EQUP_TYPE_1_Pump_RB(
	i1:= NOT( reactorB1.q6 AND reactorB2.q6 AND reactorB3.q6 AND reactorB4.q6),
	i2:= reactorB1.q6 OR reactorB2.q6 OR reactorB3.q6 OR reactorB4.q6,
	r1:= reset_Pump2_RB,
	sa1:=P201B1_DesludgePumpS2_EStopStat ,
	sa2:= ,
	sa3:=P201B1_DesludgePumpS2_LocalRemoteStat ,
	sa4:= P201B1_DesludgePumpS2_OverloadStat,
	sa5:=P201B1_DesludgePumpS2_RunStat ,
	sb1:= P201B2_DesludgePumpS2_EStopStat,
	sb2:= ,
	sb3:=P201B2_DesludgePumpS2_LocalRemoteStat ,
	sb4:= P201B2_DesludgePumpS2_OverloadStat,
	sb5:=P201B2_DesludgePumpS2_RunStat ,
	c1=> ,
	c2=> ,
	q1=>P201B1_DesludgePumpS2_RunCmd,
	q2=>P201B2_DesludgePumpS2_RunCmd ,
	e1=> );


EQUIP_TYPE_3_Valva1_RB1(
	i1:=NOT reactorB1.q1 ,
	i2:=reactorB1.q1 ,
	s1:=XV205B_SBRValveR1_CloseStat ,
	s2:=XV205B_SBRValveR1_OpenStat ,
	c1=> ,
	q1=>XV205B_SBRValveR1_CloseCmd ,
	q2=>XV205B_SBRValveR1_OpenCmd);

EQUIP_TYPE_8_MIXER_B1(
	i1:= NOT reactorB1.q2,
	i2:= reactorB1.q2,
	sa1:=M200B1A_MixerR1_EStopStat,
	sa2:=M200B1A_MixerR1_IncompleteStat ,
	sa3:=M200B1A_MixerR1_LocalRemoteStat ,
	sa4:=M200B1A_MixerR1_OverloadStat ,
	sa5:=M200B1A_MixerR1_RunStat ,
	sb1:=M200B1B_MixerR1_EStopStat,
	sb2:=M200B1B_MixerR1_IncompleteStat ,
	sb3:=M200B1B_MixerR1_LocalRemoteStat ,
	sb4:=M200B1B_MixerR1_OverloadStat ,
	sb5:=M200B1B_MixerR1_RunStat ,
	sc1:=M200B1C_MixerR1_EStopStat,
	sc2:=M200B1C_MixerR1_IncompleteStat ,
	sc3:=M200B1C_MixerR1_LocalRemoteStat ,
	sc4:=M200B1C_MixerR1_OverloadStat ,
	sc5:=M200B1C_MixerR1_RunStat ,
	c1=> ,
	q1=>M200B1A_MixerR1_RunCmd ,
	q2=>M200B1B_MixerR1_RunCmd,
	q3=>M200B1C_MixerR1_RunCmd ,
	e1=> );

EQUIP_TYPE_3_Valve2_RB1(
	i1:=NOT reactorB1.q3 ,
	i2:= reactorB1.q3,
	s1:= XV221B_LimeValveR1_CloseStat,
	s2:= XV221B_LimeValveR1_OpenStat,
	c1=> ,
	q1=>XV221B_LimeValveR1_CloseCmd ,
	q2=>XV221B_LimeValveR1_OpenCmd );

EQUIP_TYPE_3_Valve3_RB1(
	i1:=NOT reactorB1.q4 ,
	i2:= reactorB1.q4,
	s1:= XV211B_AlumValveR1_CloseStat,
	s2:= XV211B_AlumValveR1_OpenStat,
	c1=> ,
	q1=>XV211B_AlumValveR1_CloseCmd ,
	q2=>XV211B_AlumValveR1_OpenCmd );

EQUIP_TYPE_3_Valve4_RB1(
	i1:=NOT reactorB1.q5 ,
	i2:= reactorB1.q5,
	s1:=XV201B_AirBlowerValveR1_CloseStat ,
	s2:=XV201B_AirBlowerValveR1_OpenStat ,
	c1=> ,
	q1=>XV201B_AirBlowerValveR1_CloseCmd ,
	q2=>XV201B_AirBlowerValveR1_OpenCmd );

EQUIP_TYPE_9_Valve5_RB1(
	i1:= NOT reactorB1.q7 ,
	i2:=reactorB1.q7 ,
	(*s1:=XV241B_SludgeValveR1_CloseStat ,*)
	(*s2:=XV241B_SludgeValveR1_OpenStat ,*)
	c1=> ,
	q1=>XV241B_SludgeValveR1_CloseCmd ,
	q2=>XV241B_SludgeValveR1_OpenCmd );

EQUIP_TYPE_10_Dec_RB1(
	i1:=reactorB1.q8 ,
	i2:= reactorB1.q9,
	r1:= reset_dec_RB1,
	s1:= XV261B_DecanterR1_EStopStat,
	s2:= XV261B_DecanterR1_FwdStat,
	s3:= XV261B_DecanterR1_OverloadStat,
	s4:= XV261B_DecanterR1_OverloadStat,
	s5:= XV261B_DecanterR1_RvsStat,
	q1=> XV261B_DecanterR1_RvsCmd,
	q2=>XV261B_DecanterR1_FwdCmd ,
	e1=> );




EQUIP_TYPE_3_Valva1_RB2(
	i1:=NOT reactorB2.q1 ,
	i2:=reactorB2.q1 ,
	s1:=XV206B_SBRValveR2_CloseStat ,
	s2:=XV206B_SBRValveR2_OpenStat ,
	c1=> ,
	q1=>XV206B_SBRValveR2_CloseCmd ,
	q2=>XV206B_SBRValveR2_OpenCmd);

EQUIP_TYPE_8_MIXER_B2(
	i1:= NOT reactorB2.q2,
	i2:= reactorB2.q2,
	sa1:=M200B2A_MixerR2_EStopStat,
	sa2:=M200B2A_MixerR2_IncompleteStat ,
	sa3:=M200B2A_MixerR2_LocalRemoteStat ,
	sa4:=M200B2A_MixerR2_OverloadStat ,
	sa5:=M200B2A_MixerR2_RunStat ,
	sb1:=M200B2B_MixerR2_EStopStat,
	sb2:=M200B2B_MixerR2_IncompleteStat ,
	sb3:=M200B2B_MixerR2_LocalRemoteStat ,
	sb4:=M200B2B_MixerR2_OverloadStat ,
	sb5:=M200B2B_MixerR2_RunStat ,
	sc1:=M200B2C_MixerR2_EStopStat,
	sc2:=M200B2C_MixerR2_IncompleteStat ,
	sc3:=M200B2C_MixerR2_LocalRemoteStat ,
	sc4:=M200B2C_MixerR2_OverloadStat ,
	sc5:=M200B2C_MixerR2_RunStat ,
	c1=> ,
	q1=>M200B2A_MixerR2_RunCmd ,
	q2=>M200B2B_MixerR2_RunCmd,
	q3=>M200B2C_MixerR2_RunCmd ,
	e1=> );

EQUIP_TYPE_3_Valve2_RB2(
	i1:=NOT reactorB2.q3 ,
	i2:= reactorB2.q3,
	s1:= XV222B_LimeValveR2_CloseStat,
	s2:= XV222B_LimeValveR2_OpenStat,
	c1=> ,
	q1=>XV222B_LimeValveR2_CloseCmd ,
	q2=>XV222B_LimeValveR2_OpenCmd );

EQUIP_TYPE_3_Valve3_RB2(
	i1:=NOT reactorB2.q4 ,
	i2:= reactorB2.q4,
	s1:= XV212B_AlumValveR2_CloseStat,
	s2:= XV212B_AlumValveR2_OpenStat,
	c1=> ,
	q1=>XV212B_AlumValveR2_CloseCmd ,
	q2=>XV212B_AlumValveR2_OpenCmd );

EQUIP_TYPE_3_Valve4_RB2(
	i1:=NOT reactorB2.q5 ,
	i2:= reactorB2.q5,
	s1:=XV202B_AirBlowerValveR2_CloseStat ,
	s2:=XV202B_AirBlowerValveR2_OpenStat ,
	c1=> ,
	q1=>XV202B_AirBlowerValveR2_CloseCmd ,
	q2=>XV202B_AirBlowerValveR2_OpenCmd );


EQUIP_TYPE_9_Valve5_RB2(
	i1:= NOT reactorB2.q7 ,
	i2:=reactorB2.q7 ,
	(*s1:=XV242B_SludgeValveR2_CloseStat ,*)
	(*s2:=XV242B_SludgeValveR2_OpenStat ,*)
	c1=> ,
	q1=>XV242B_SludgeValveR2_CloseCmd ,
	q2=>XV242B_SludgeValveR2_OpenCmd );

EQUIP_TYPE_10_Dec_RB2(
	i1:=reactorB2.q8 ,
	i2:= reactorB2.q9,
	r1:= reset_dec_RB2,
	s1:= XV262B_DecanterR2_EStopStat,
	s2:= XV262B_DecanterR2_FwdStat,
	s3:= XV262B_DecanterR2_OverloadStat,
	s4:= XV262B_DecanterR2_OverloadStat,
	s5:= XV262B_DecanterR2_RvsStat,
	q1=> XV262B_DecanterR2_RvsCmd,
	q2=>XV262B_DecanterR2_FwdCmd ,
	e1=> );




EQUIP_TYPE_3_Valva1_RB3(
	i1:=NOT reactorB3.q1 ,
	i2:=reactorB3.q1 ,
	s1:=XV207B_SBRValveR3_CloseStat ,
	s2:=XV207B_SBRValveR3_OpenStat ,
	c1=> ,
	q1=>XV207B_SBRValveR3_CloseCmd ,
	q2=>XV207B_SBRValveR3_OpenCmd);

EQUIP_TYPE_8_MIXER_B3(
	i1:= NOT reactorB3.q2,
	i2:= reactorB3.q2,
	sa1:=M200B3A_MixerR3_EStopStat,
(*	sa2:=M200B3A_MixerR3_IncompleteStat ,*)
	sa3:=M200B3A_MixerR3_LocalRemoteStat ,
	sa4:=M200B3A_MixerR3_OverloadStat ,
	sa5:=M200B3A_MixerR3_RunStat ,
	sb1:=M200B3B_MixerR3_EStopStat,
	sb2:=M200B3B_MixerR3_IncompleteStat ,
	sb3:=M200B3B_MixerR3_LocalRemoteStat ,
	sb4:=M200B3B_MixerR3_OverloadStat ,
	sb5:=M200B3B_MixerR3_RunStat ,
	sc1:=M200B3C_MixerR3_EStopStat,
	sc2:=M200B3C_MixerR3_IncompleteStat ,
	sc3:=M200B3C_MixerR3_LocalRemoteStat ,
	sc4:=M200B3C_MixerR3_OverloadStat ,
	sc5:=M200B3C_MixerR3_RunStat ,
	c1=> ,
	q1=>M200B3A_MixerR3_RunCmd ,
	q2=>M200B3B_MixerR3_RunCmd,
	q3=>M200B3C_MixerR3_RunCmd ,
	e1=> );

EQUIP_TYPE_3_Valve2_RB3(
	i1:=NOT reactorB3.q3 ,
	i2:= reactorB3.q3,
	s1:= XV223B_LimeValveR3_CloseStat,
	s2:= XV223B_LimeValveR3_OpenStat,
	c1=> ,
	q1=>XV223B_LimeValveR3_CloseCmd ,
	q2=>XV223B_LimeValveR3_OpenCmd );

EQUIP_TYPE_3_Valve3_RB3(
	i1:=NOT reactorB3.q4 ,
	i2:= reactorB3.q4,
	s1:= XV213B_AlumValveR3_CloseStat,
	s2:= XV213B_AlumValveR3_OpenStat,
	c1=> ,
	q1=>XV213B_AlumValveR3_CloseCmd ,
	q2=>XV213B_AlumValveR3_OpenCmd );

EQUIP_TYPE_3_Valve4_RB3(
	i1:=NOT reactorB3.q5 ,
	i2:= reactorB3.q5,
	s1:=XV203B_AirBlowerValveR3_CloseStat ,
	s2:=XV203B_AirBlowerValveR3_OpenStat ,
	c1=> ,
	q1=>XV203B_AirBlowerValveR3_CloseCmd ,
	q2=>XV203B_AirBlowerValveR3_OpenCmd );


EQUIP_TYPE_9_Valve5_RB3(
	i1:= NOT reactorB3.q7 ,
	i2:=reactorB3.q7 ,
	(*s1:=XV243B_SludgeValveR3_CloseStat ,*)
	(*s2:=XV243B_SludgeValveR3_OpenStat ,*)
	c1=> ,
	q1=>XV243B_SludgeValveClosedR3_CloseCmd ,
	q2=>XV243B_SludgeValveR3_OpenCmd );

EQUIP_TYPE_10_Dec_RB3(
	i1:=reactorB3.q8 ,
	i2:= reactorB3.q9,
	r1:= reset_dec_RB3,
	s1:= XV263B_DecanterR3_EStopStat,
	s2:= XV263B_DecanterR3_FwdStat,
	s3:= XV263B_DecanterR3_OverloadStat,
	s4:= XV263B_DecanterR3_OverloadStat,
	s5:= XV263B_DecanterR3_RvsStat,
	q1=> XV263B_DecanterR3_RvsCmd,
	q2=>XV263B_DecanterR3_FwdCmd ,
	e1=> );



EQUIP_TYPE_3_Valva1_RB4(
	i1:=NOT reactorB4.q1 ,
	i2:=reactorB4.q1 ,
	s1:=XV208B_SBRValveR4_CloseStat ,
	s2:=XV208B_SBRValveR4_OpenStat ,
	c1=> ,
	q1=>XV208B_SBRValveR4_CloseCmd ,
	q2=>XV208B_SBRValveR4_OpenCmd);

EQUIP_TYPE_8_MIXER_B4(
	i1:= NOT reactorB4.q2,
	i2:= reactorB4.q2,
	(*sa1:=M200B4A_MixerR4_EStopStat,*)
	sa2:=M200B4A_MixerR4_IncompleteStat ,
	sa3:=M200B4A_MixerR4_LocalRemoteStat ,
	sa4:=M200B4A_MixerR4_OverloadStat ,
	sa5:=M200B4A_MixerR4_RunStat ,
	(*sb1:=M200B4B_MixerR4_EStopStat,*)
	sb2:=M200B4B_MixerR4_IncompleteStat ,
	sb3:=M200B4B_MixerR4_LocalRemoteStat ,
	sb4:=M200B4B_MixerR4_OverloadStat ,
	sb5:=M200B4B_MixerR4_RunStat ,
	(*sc1:=M200B4C_MixerR4_EStopStat,*)
	sc2:=M200B4C_MixerR4_IncompleteStat ,
	sc3:=M200B4C_MixerR4_LocalRemoteStat ,
	sc4:=M200B4C_MixerR4_OverloadStat ,
	sc5:=M200B4C_MixerR4_RunStat ,
	c1=> ,
	q1=>M200B4A_MixerR4_RunCmd ,
	q2=>M200B4B_MixerR4_RunCmd,
	q3=>M200B4C_MixerR4_RunCmd ,
	e1=> );

EQUIP_TYPE_3_Valve2_RB4(
	i1:=NOT reactorB4.q3 ,
	i2:= reactorB4.q3,
	s1:= XV224B_LimeValveR4_CloseStat,
	s2:= XV224B_LimeValveR4_OpenStat,
	c1=> ,
	q1=>XV224B_LimeValveR4_CloseCmd ,
	q2=>XV224B_LimeValveR4_OpenCmd );

EQUIP_TYPE_3_Valve3_RB4(
	i1:=NOT reactorB4.q4 ,
	i2:= reactorB4.q4,
	s1:= XV214B_AlumValveR4_CloseStat,
	s2:= XV214B_AlumValveR4_OpenStat,
	c1=> ,
	q1=>XV214B_AlumValveR4_CloseCmd ,
	q2=>XV214B_AlumValveR4_OpenCmd );

EQUIP_TYPE_3_Valve4_RB4(
	i1:=NOT reactorB4.q5 ,
	i2:= reactorB4.q5,
	s1:=XV204B_AirBlowerValveR4_CloseStat ,
	s2:=XV204B_AirBlowerValveR4_OpenStat ,
	c1=> ,
	q1=>XV204B_AirBlowerValveR4_CloseCmd ,
	q2=>XV204B_AirBlowerValveR4_OpenCmd );

EQUIP_TYPE_9_Valve5_RB4(
	i1:= NOT reactorB4.q7 ,
	i2:=reactorB4.q7 ,
	(*s1:=XV244B_SludgeValveR4_CloseStat ,*)
	(*s2:=XV244B_SludgeValveR4_OpenStat ,*)
	c1=> ,
	q1=>XV244B_SludgeValveR4_CloseCmd ,
	q2=>XV244B_SludgeValveR4_OpenCmd );

EQUIP_TYPE_10_Dec_RB4(
	i1:=reactorB4.q8 ,
	i2:= reactorB4.q9,
	r1:= reset_dec_RB4,
	s1:= XV264B_DecanterR4_EStopStat,
	s2:= XV264B_DecanterR4_FwdStat,
	s3:= XV264B_DecanterR4_OverloadStat,
	s4:= XV264B_DecanterR4_OverloadStat,
	s5:= XV264B_DecanterR4_RvsStat,
	q1=> XV264B_DecanterR4_RvsCmd,
	q2=>XV264B_DecanterR4_FwdCmd ,
	e1=> );
END_ACTION

(* POU INLET, ST *)
FUNCTION_BLOCK INLET
VAR_INPUT
(*inlet*)
	i1: BOOL;
	i3: BOOL;
	i2: BOOL;
	i4: BOOL;

(*MIXER*)

	i5: BOOL;
	i6: BOOL;

(*penstock*)
	r1: BOOL; (*rs1*)
	i7: BOOL; (*ps open*)
	i8: BOOL;	(*ps open*)
	i10: BOOL;
	i9: BOOL;
	i11: BOOL;
	s1: BOOL;
	s2: BOOL;
	s3: BOOL;
	s4: BOOL;

(* sbr transfer *)
	i12: BOOL;
	i13: BOOL;


	i14: BOOL;
END_VAR
VAR_OUTPUT

(*inlet*)
	q1: BOOL;
	q2: BOOL;

(*MIXER*)

	q3: BOOL;
	q4: BOOL;

(*penstock*)
	q5: BOOL; (*ps1*)
	q6: BOOL; (*ps2*)
	q7: BOOL;
	q8: BOOL;
	q10: BOOL;
	q9: BOOL;
	q11: BOOL;
	q12: BOOL;
	q13: BOOL;
	q14: BOOL;
	q15: BOOL;
	q16: BOOL;
	q17: BOOL;
	q18: BOOL;
	q19: BOOL;
	q20: BOOL;
(* Grit Removal*)

	q21: BOOL;
	q22: BOOL;
	q23: BOOL;
	q24: BOOL;
	q25:BOOL;
	q26:BOOL;

(* sbr transfer *)

	q27: BOOL;
	q28: BOOL;

END_VAR
VAR
(*inlet*)
	m1: BOOL;
	ton1: TON;

(*MIXER*)


(*penstock*)
	penstock: INT;
	FailedGroupA: BOOL;
	FailedGroupB: BOOL;
	m2: BOOL;
	TP1: TP;
	m3: BOOL;
	TON2: TON;
	TON3: TON;
	TOF1: TOF;
	TON4 : TON;
	mr: BOOL;
	F_TRIG1: F_TRIG;
	R_TRIG1: R_TRIG;
	m4 : BOOL;
	TON5: TON;

END_VAR



(*
CASE penstock OF
0:
	q5 := TRUE;
	q6 := FALSE;
	IF FailedGroupA OR m2 THEN
		penstock := 1;
	END_IF
1 :
 	q6 := TRUE;
	IF FailedGroupB THEN
		penstock := 2;
	ELSIF i8 THEN
		penstock := 3;
	END_IF
2 :
	q5 := FALSE;
	q6 := FALSE;
	IF r1 THEN
		penstock := 0;
	END_IF
3:
	q6 := TRUE;
	q5 := FALSE;
	IF FailedGroupB OR m2 THEN
		penstock := 4;
	END_IF
4 :
	q6 := TRUE;
	IF FailedGroupA THEN
		penstock := 2;
	ELSIF i7 THEN
		penstock := 0;
	END_IF
END_CASE*)
(*EQ Pump*)
q1 := NOT i1 OR i3 OR m1;
q2 := i2 AND NOT i3 AND NOT m1;
ton1(IN:=i4 , PT:=t#5m , Q=>m1 , ET=> );

(*Mixer*)
q3 := NOT i5;
q4 := i6;


(*screen*)
FailedGroupA := s1 OR s2;
FailedGroupB := s3 OR s4;

m4 := ((NOT m4 AND (FailedGroupA OR m2)) OR m4) AND NOT((m4 AND (FailedGroupB OR m2)) OR r1);
q5 := (NOT m4 OR q5) AND NOT(( m4 AND i8) OR mr) ;
q6 := (m4 OR q6) AND NOT ((NOT m4 AND i7) OR mr);
mr := (mr OR (FailedGroupA AND FailedGroupB)) AND NOT r1;

TOF1(IN:=i11 , PT:=T#2m , Q=>i9 , ET=> );

F_TRIG1(CLK:=m4 );
R_TRIG1(CLK:=m4 );
TP1(IN:=(F_TRIG1.Q OR R_TRIG1.Q) , PT:= T#5m , Q=>m3 , ET=> );
m2 := i10 AND NOT m3;

TON4(IN:=NOT i9 OR NOT(q5 OR q6) , PT:=T#5m , Q=>q7 , ET=> );
TON2(IN:= i9 AND (q5 OR q6), PT := T#1h, Q=> q8);

TON3(IN:=q7,PT:=T#5m,Q=>q9);
q10 := q8;

q11 := q9;
q12 := q10;

q13 := NOT (i9 AND Q5);
q14 := (i9 AND Q5);

q15 := NOT(i9 AND q6);
q16 := (i9 AND q6);

q17 := q13;
q18 := q14;

q19 := q15;
q20 :=q18;

(*Grit Removal*)
q21 := i7;
q22 := i8;

q23 := NOT i9;
q24 := i9;

TON5(IN:= NOT i9, PT:=T#5m , Q=>q25 );
q26 := i9;


(*sbr transfer*)
q27  := NOT i12;
q28 := i13 AND i14;
END_FUNCTION_BLOCK

(* POU EQUP_TYPE_1, ST *)
FUNCTION_BLOCK EQUP_TYPE_1
VAR_INPUT
	i1 : BOOL;
	i2 : BOOL;
	r1 : BOOL;

	sa1 : BOOL;
	sa2 : BOOL;
	sa3 : BOOL;
	sa4 : BOOL;
	sa5 : BOOL;

	sb1 : BOOL;
	sb2 : BOOL;
	sb3 : BOOL;
	sb4 : BOOL;
	sb5 : BOOL;
END_VAR
VAR_OUTPUT
	c1 : BOOL;
	c2 :BOOL;
	q1 : BOOL;
	q2 : BOOL;
	e1 : BOOL;
END_VAR
VAR
	toggle : INT;
END_VAR
c1 := (i2 OR c1) AND NOT i1;
e1 :=(( (sa2 OR sa4 OR sa1) AND (sb2 OR sb4 OR sb1)) OR e1) AND NOT r1;

CASE toggle OF
0:
	c2 := TRUE;
	IF e1 THEN
		toggle := 3;
	ELSIF sa2 OR sa4 OR sa1 THEN
		toggle := 1;
	END_IF
1:
	c2 := FALSE;
	IF e1 THEN
		toggle := 3;
	ELSIF  sb2 OR sb4 OR sb1 THEN
		toggle := 0;
	END_IF
3:
	IF r1 THEN
		toggle := 0;
	END_IF

END_CASE

q1 := c1 AND NOT c2;
q2 := c1 AND c2;
END_FUNCTION_BLOCK

(* POU EQUIP_TYPE_2, ST *)
FUNCTION_BLOCK EQUIP_TYPE_2
VAR_INPUT
	i1 : BOOL;
	i2 : BOOL;

	sa1 : BOOL;
	sa2 : BOOL;
	sa3 : BOOL;
	sa4 : BOOL;
	sa5 : BOOL;

	sb1 : BOOL;
	sb2 : BOOL;
	sb3 : BOOL;
	sb4 : BOOL;
	sb5 : BOOL;
END_VAR
VAR_OUTPUT
	c1 : BOOL;
	q1 : BOOL;
	q2 : BOOL;
	e1 : BOOL;
END_VAR
VAR
END_VAR
c1 := (i2 OR c1) AND NOT i1;
e1 :=(( (sa2 OR sa4 OR sa1) AND (sb2 OR sb4 OR sb1)));
q1 := c1;
q2 := c1;
END_FUNCTION_BLOCK

(* POU EQUIP_TYPE_3, ST *)
FUNCTION_BLOCK EQUIP_TYPE_3
VAR_INPUT
	i1:BOOL;
	i2 : BOOL;
	s1:BOOL;
	s2:BOOL;
	s3:BOOL;
	s4:BOOL;
END_VAR
VAR_OUTPUT
	c1 : BOOL;
	q1: BOOL;
	q2: BOOL;
END_VAR
VAR
END_VAR
c1 := (i2 OR c1) AND NOT i1;
q1 := NOT c1;
q2 := c1;
END_FUNCTION_BLOCK

(* POU EQUIP_TYPE_4, ST *)
FUNCTION_BLOCK EQUIP_TYPE_4
(*
	sa1:= F101B2_FineScr_EStopStat,
	sa2:= F101B2_FineScr_LocalRemoteStat,
	sa3:= F101B2_FineScr_OverloadStat,
	sa4:= F101B2_FineScr_RunStat,
*)
VAR_INPUT
	i1 : BOOL;
	i2 : BOOL;

	sa1 : BOOL;
	sa2 : BOOL;
	sa3 : BOOL;
	sa4 : BOOL;

END_VAR
VAR_OUTPUT
	c1 : BOOL;
	q1 : BOOL;
	e1 : BOOL;
END_VAR
VAR
END_VAR
c1 := (i2 OR c1) AND NOT i1;
e1 :=( ( sa3 OR sa1));
q1 := c1;
END_FUNCTION_BLOCK

(* POU EQUIP_TYPE_5, ST *)
FUNCTION_BLOCK EQUIP_TYPE_5
VAR_INPUT
	i1 : BOOL;
	i2 : BOOL;

	sa1 : BOOL;
	sa2 : BOOL;

END_VAR
VAR_OUTPUT
	c1 : BOOL;
	q1 : BOOL;
	e1 : BOOL;
END_VAR
VAR
END_VAR
c1 := (i2 OR c1) AND NOT i1;
q1 := c1;
END_FUNCTION_BLOCK

(* POU EQUIP_TYPE_6, ST *)
FUNCTION_BLOCK EQUIP_TYPE_6 (*NEED TO IMPLEMENT TIMER*)
VAR_INPUT
	i1 : BOOL;
	i2 : BOOL;

	sa1 : BOOL;
	sa2 : BOOL;

END_VAR
VAR_OUTPUT
	c1 : BOOL;
	q1 : BOOL;
	e1 : BOOL;
END_VAR
VAR
END_VAR
c1 := (i2 OR c1) AND NOT i1;
q1 := c1;
END_FUNCTION_BLOCK

(* POU EQUP_TYPE_7, ST *)
FUNCTION_BLOCK EQUP_TYPE_7 (* cycle not done yet *)
VAR_INPUT
	i1 : BOOL;
	i2 : BOOL;
	r1 : BOOL;

	sa1 : BOOL;
	sa2 : BOOL;
	sa3 : BOOL;
	sa4 : BOOL;
	sa5 : BOOL;

	sb1 : BOOL;
	sb2 : BOOL;
	sb3 : BOOL;
	sb4 : BOOL;
	sb5 : BOOL;
END_VAR
VAR_OUTPUT
	c1 : BOOL;
	c2 :BOOL;
	q1 : BOOL;
	q2 : BOOL;
	e1 : BOOL;
END_VAR
VAR
	toggle : INT;
END_VAR
c1 := (i2 OR c1) AND NOT i1;
e1 :=(( (sa2 OR sa4 OR sa1) AND (sb2 OR sb4 OR sb1)) OR e1) AND NOT r1;

CASE toggle OF
0:
	c2 := TRUE;
	IF e1 THEN
		toggle := 3;
	ELSIF sa2 OR sa4 OR sa1 THEN
		toggle := 1;
	END_IF
1:
	c2 := FALSE;
	IF e1 THEN
		toggle := 3;
	ELSIF  sb2 OR sb4 OR sb1 THEN
		toggle := 0;
	END_IF
3:
	IF r1 THEN
		toggle := 0;
	END_IF

END_CASE

q1 := c1 AND NOT c2;
q2 := c1 AND c2;
END_FUNCTION_BLOCK

(* POU Chemical_new, ST *)
FUNCTION_BLOCK Chemical_new
VAR_INPUT
	iA1: BOOL;
	iA2: BOOL;
	iA3: BOOL;
	iA4: BOOL;
	rA1: BOOL;

	iB1: BOOL;
	iB2: BOOL;
	iB3: BOOL;
	iB4: BOOL;
	rB1: BOOL;

	iC1: BOOL;
	iC2: BOOL;
	iC3: BOOL;
	iC4: BOOL;
	rC1: BOOL;


	iqA2: BOOL;
	iqB2: BOOL;
	iqC2: BOOL;


	iLRA: BOOL;
	iLRB: BOOL;

	iAop1: BOOL;
	iAop2: BOOL;
	iAop3: BOOL;
	iAop4: BOOL;



	iAlss1: BOOL;
	iAlss2: BOOL;
	iAlss3: BOOL;
	iAlss4: BOOL;

	iasbrA: BOOL; (*sbr alum vale*)
	iasbrB: BOOL;

	iCop1 : BOOL;
	iCop2 : BOOL;
	ilssC1 : BOOL;
	ilssC2 : BOOL;

	itpm : BOOL;
	itpC : BOOL;
	itpCh : BOOL;

	ilssch1: BOOL;
	ilssch2: BOOL;
	ilssch3: BOOL;

	iChop1: BOOL;
	iChop2: BOOL;
	iChop3: BOOL;

	irdAB : BOOL;



END_VAR
VAR_OUTPUT
	qA1: BOOL;
	qA2: BOOL;
	qA3: BOOL;
	eA1: BOOL;

	qB1: BOOL;
	qB2: BOOL;
	qB3: BOOL;
	eB1: BOOL;

	qC1: BOOL;
	qC2: BOOL;
	qC3: BOOL;
	eC1: BOOL;

	qD1: BOOL;
	qD2: BOOL;
	qD3: BOOL;
	eD1: BOOL;

	qCir: BOOL;

	qLA: BOOL;
	qLB: BOOL;

	qP1: BOOL;
	qP2: BOOL;

	qP3: BOOL;
	qP4: BOOL;

	qtA1: BOOL;
	qtC1: BOOL;
	qtCH1: BOOL;

	qdsp : BOOL;


END_VAR
VAR
	tank_lime_A: tanks;
	tank_lime_B: tanks;
	tank_lime_C: tanks;


	alumtankstat: BOOL;
	limetankstat: BOOL;
	caustictankstat: BOOL;
	chlorintankstat: BOOL;

END_VAR
tank_lime_A(
	LSLL:=iA1 ,
	LSL:= iA2,
	LSH:= iA3,
	LSHH:=iA4 ,
	reset:= rA1,
	fill=> qA1,
	valve=> qA2,
	mixer=> qA3,
	alarm=>eA1 );

tank_lime_B(
	LSLL:=iB1 ,
	LSL:= iB2,
	LSH:= iB3,
	LSHH:=iB4 ,
	reset:= rB1,
	fill=> qB1,
	valve=> qB2,
	mixer=> qB3,
	alarm=>eB1 );

tank_lime_C(
	LSLL:=iC1 ,
	LSL:= iC2,
	LSH:= iC3,
	LSHH:=iC4 ,
	reset:= rC1,
	fill=> qC1,
	valve=> qC2,
	mixer=> qC3,
	alarm=>eC1 );


qCir := TRUE;

qLA := iLRA;
qLB := iLRB;

limetankstat;


qP1 :=iLRA AND (iqA2 OR iqB2 OR iqC2);
qP2 := iLRA AND (iqA2 OR iqB2 OR iqC2);

alumtankstat := (iAlss1 AND iAop1) OR (iAlss2 AND iAop2) OR (iAlss3 AND iAop3) OR (iAlss4 AND iAop4);

(*Alum tank*)
qP3 := iasbrA AND alumtankstat;
qP4 := iasbrB AND alumtankstat;

(*alum tank tertiary*)
qtA1 := itpm AND alumtankstat;


(*caustic*)
caustictankstat := (ilssc1 AND iCop1) OR (ilssc2 AND iCop2);
qtC1 := caustictankstat AND itpc;

(*clorin*)
chlorintankstat := (ilssch1 AND iChop1) OR (ilssch2 AND iChop2) OR (ilssch3 AND iChop3);
qtCH1 := chlorintankstat AND itpCh;

(*effuent disinfection*)
qdsp := irdAB AND chlorintankstat;
END_FUNCTION_BLOCK

(* POU tanks, ST *)
FUNCTION_BLOCK tanks
VAR_INPUT
	LSLL: BOOL;
	LSL: BOOL;
	LSH: BOOL;
	LSHH: BOOL;

	reset: BOOL;

END_VAR
VAR_OUTPUT

	fill: BOOL;
	valve: BOOL;
	mixer: BOOL;
	alarm: BOOL;
END_VAR
VAR
	tank: INT;
END_VAR
IF NOT  LSLL THEN
	fill := TRUE;
ELSIF LSHH THEN
	fill:= FALSE;
END_IF

valve := FALSE;
alarm := FALSE;
CASE tank OF
0: IF lsh THEN
	tank := 1;
	alarm := TRUE;
      END_IF
1:
	IF reset THEN
		alarm := FALSE;
		valve := TRUE;
		tank := 2;
	END_IF
2 :
	IF NOT lsll THEN
		tank := 0;
	END_IF
END_CASE

IF LSL THEN
	mixer := TRUE;
ELSIF NOT lsll THEN
	mixer := FALSE;
END_IF
END_FUNCTION_BLOCK

(* POU Reactor, ST *)
FUNCTION_BLOCK Reactor
VAR_INPUT
	op: BOOL;
	res_fill: BOOL;
	i1: BOOL;
	alum_time: TIME := T#5s;
	res_aeration: BOOL;
	ph1: REAL;
	res_decanting: BOOL;
	r1: BOOL;
	i2: BOOL;
	i3: BOOL;
	i4: BOOL;
END_VAR
VAR_OUTPUT
	req_fill: BOOL;
	q1: BOOL;
	q2: BOOL;
	q4: BOOL;
	q3: BOOL;
	q5: BOOL;
	q6: BOOL;
	req_aeration: BOOL;
	e1: BOOL;
	q7: BOOL;
	q8: BOOL;
	m1:BOOL;
	req_settle: BOOL;
	req_decanting: BOOL;
	q9: BOOL;
END_VAR
VAR
	seq: INT;
	TON1: TON;
	TP1: TP;
	TON2: TON;
	TON3: TON;
	decanting_done: BOOL;
	start_decanter: BOOL;
	TON4: TON;
	decanter: INT;
	TP2: TP;
	TP3: TP;
END_VAR
req_fill := FALSE;
req_aeration := FALSE;
req_settle:= FALSE;
req_decanting := FALSE;
start_decanter := FALSE;
q1 := FALSE;
q2 := FALSE;
q3 := FALSE;
q4 := FALSE;
q5 := FALSE;

q6 := FALSE;
q7 := FALSE;

q8 := FALSE;
q9 := FALSE;
CASE seq OF
0:
	IF op THEN
		seq := 1;
	END_IF
1:
IF op THEN
	req_fill := TRUE;
	q1 := res_fill;
	q2 := TRUE;

	IF i1 THEN
		seq := 2;
	END_IF
ELSE
	seq := 0;
END_IF
2:
IF op THEN
	req_aeration := TRUE;
	IF res_aeration THEN
		TON2(IN:= TRUE,PT:=T#3.5h , Q=> , ET=> );

		TON1(IN:= TRUE, PT:=T#2h , Q=> e1, ET=> );
		TP1(IN:=TON1.Q AND r1 , PT:=alum_time , Q=>q4 , ET=> );
		q5 := TRUE;
		m1 := ((m1 OR (ph1 <= 5)) AND ph1 > 7.5);
		q3 := m1;
		IF ton2.Q THEN
			TON2(IN:= FALSE,PT:=T#3.5h , Q=> , ET=> );

			TON1(IN:= FALSE, PT:=T#2h , Q=> e1, ET=> );
			TP1(IN:=FALSE , PT:=alum_time , Q=>q4 , ET=> );
			seq := 3;
		END_IF
	END_IF

ELSE
	seq := 0;
	TON2(IN:= FALSE,PT:=T#3.5h , Q=> , ET=> );

	TON1(IN:= FALSE, PT:=T#2h , Q=> e1, ET=> );
	TP1(IN:=FALSE , PT:=alum_time , Q=>q4 , ET=> );
END_IF
3:
IF op THEN
	req_settle  := TRUE;
	TON3(IN:=TRUE ,  PT:=T#1.5h);
	IF ton3.Q THEN
		seq:= 4;
		TON3(IN:=FALSE ,  PT:=T#1.5h);
	END_IF
ELSE
	seq:= 0;
	TON3(IN:=FALSE ,  PT:=T#1.5h);
END_IF

4:
IF op THEN
 	req_decanting := TRUE;
	IF res_decanting THEN
		start_decanter := TRUE;
	END_IF
	IF decanting_done THEN
		seq := 0;
		TON4(IN:=FALSE ,  PT:=T#3606s);
	END_IF
	TON4(IN:=TRUE, PT:=T#3606s);
	IF ((TON4.ET < T#15m) OR (TON4.ET > T#45m)) AND NOT i2 THEN
		q6 := TRUE;
		q7 := TRUE;
	END_IF
ELSE
	seq:=0;
END_IF
END_CASE


decanting_done := FALSE;
CASE decanter OF
0:
	q8 := NOT i3;
	q9 := FALSE;

	IF i3 AND start_decanter THEN
		decanter := 1;
	END_IF

1:
	q8 := FALSE;
	IF start_decanter THEN
		TP2(IN:=TRUE , PT:=T#45s , Q=> q9, ET=> );
		IF NOT TP2.Q OR i4 THEN
			decanter := 2;
			TP2(IN:=FALSE , PT:=T#45s , Q=> q9, ET=> );
		END_IF
	END_IF
2:
	IF start_decanter THEN
		TP3(IN:=TRUE , PT:=T#5s , Q=> q9, ET=> );
		IF i4 THEN
			decanter := 0;
			TP3(IN:=FALSE , PT:=T#5s , Q=> q9, ET=> );
			decanting_done := TRUE;
		ELSIF (NOT TP3.Q) THEN
			decanter := 1;
			TP3(IN:=FALSE , PT:=T#5s , Q=> q9, ET=> );
		END_IF
	END_IF
END_CASE
END_FUNCTION_BLOCK

(* POU Fill_selector, ST *)
FUNCTION_BLOCK Fill_selector
VAR_INPUT
	i1: BOOL;
	i2: BOOL;
	i3: BOOL;
	i4: BOOL;
END_VAR
VAR_OUTPUT
	q1: BOOL;
	q2: BOOL;
	q3: BOOL;
	q4: BOOL;
	c1 : BOOL;
END_VAR
VAR
	ireactor: INT;
END_VAR
q1 := q2 := q3 := q4 := FALSE;

CASE ireactor OF
0:
	IF NOT i1 THEN
		ireactor := 1;
	END_IF
	q1 := TRUE;
1:
	IF NOT i2 THEN
		ireactor := 2;
	END_IF
	q2 := TRUE;
2:
	IF NOT i3 THEN
		ireactor := 3;
	END_IF
	q3 := TRUE;
3:
	IF NOT i4 THEN
		ireactor := 0;
	END_IF
	q4 := TRUE;
END_CASE

c1 := i1 OR i2 OR i3 OR i4;
END_FUNCTION_BLOCK

(* POU blower_selector, ST *)
FUNCTION_BLOCK blower_selector
VAR_INPUT
	i1 :BOOL;
	i2: BOOL;
	i3 : BOOL;
	i4 : BOOL;
	available : INT;
END_VAR
VAR_OUTPUT
	q1 : BOOL;
	q2 : BOOL;
	q3 : BOOL;
	q4 : BOOL;
	taken : INT;
END_VAR
VAR
	request: ARRAY [1..4] OF BOOL;
	respond: ARRAY [1..4] OF BOOL;
	b: INT;
	a: INT;
END_VAR
request[a];
respond[b];
taken;
available;


request[1] := i1;
request[2] := i2;
request[3] := i3;
request[4] := i4;
FOR a:= 1 TO 4 DO
IF request[a] AND NOT respond[a] THEN
	IF available - taken > 0 THEN
		respond[a] := TRUE;
		taken := taken+ 1;
	END_IF
END_IF
END_FOR

FOR b:=1 TO 4 DO
IF respond[b] THEN
	IF NOT request[b] THEN
		respond[b] := FALSE;
		taken := taken -1;
		IF taken < 0 THEN
			taken := 0;
		END_IF
	END_IF
END_IF
END_FOR
q1 := respond[1];
q2 := respond[2];
q3 := respond[3];
q4 := respond[4];
END_FUNCTION_BLOCK

(* POU Decant_selector, ST *)
FUNCTION_BLOCK Decant_selector
VAR_INPUT
	i1: BOOL;
	i2: BOOL;
	i3: BOOL;
	i4: BOOL;
END_VAR
VAR_OUTPUT
	q1: BOOL;
	q2: BOOL;
	q3: BOOL;
	q4: BOOL;
	c1: BOOL;
END_VAR
VAR
	ireactor: INT;
END_VAR
q1 := q2 := q3 := q4 := FALSE;

CASE ireactor OF
0:
	IF NOT i1 THEN
		ireactor := 1;
	END_IF
	q1 := TRUE;
1:
	IF NOT i2 THEN
		ireactor := 2;
	END_IF
	q2 := TRUE;
2:
	IF NOT i3 THEN
		ireactor := 3;
	END_IF
	q3 := TRUE;
3:
	IF NOT i4 THEN
		ireactor := 0;
	END_IF
	q4 := TRUE;
END_CASE

c1 := i1 OR i2 OR i3 OR i4;
END_FUNCTION_BLOCK

(* POU EQUIP_TYPE_9, ST *)
FUNCTION_BLOCK EQUIP_TYPE_9 (*same as type 3 with lesser input*)
VAR_INPUT
	i1:BOOL;
	i2 : BOOL;
	s1:BOOL;
	s2:BOOL;
END_VAR
VAR_OUTPUT
	c1 : BOOL;
	q1: BOOL;
	q2: BOOL;
END_VAR
VAR
END_VAR
c1 := (i2 OR c1) AND NOT i1;
q1 := NOT c1;
q2 := c1;
END_FUNCTION_BLOCK

(* POU EQUIP_TYPE_8, ST *)
FUNCTION_BLOCK EQUIP_TYPE_8
VAR_INPUT
	i1 : BOOL;
	i2 : BOOL;

	sa1 : BOOL;
	sa2 : BOOL;
	sa3 : BOOL;
	sa4 : BOOL;
	sa5 : BOOL;

	sb1 : BOOL;
	sb2 : BOOL;
	sb3 : BOOL;
	sb4 : BOOL;
	sb5 : BOOL;

	sc1 : BOOL;
	sc2 : BOOL;
	sc3 : BOOL;
	sc4 : BOOL;
	sc5 : BOOL;
END_VAR
VAR_OUTPUT
	c1 : BOOL;
	q1 : BOOL;
	q2 : BOOL;
	q3 : BOOL;
	e1 : BOOL;
END_VAR
VAR
END_VAR
c1 := (i2 OR c1) AND NOT i1;
e1 :=(( (sa2 OR sa4 OR sa1) AND (sb2 OR sb4 OR sb1)AND (sc2 OR sc4 OR sc1)));
q1 := c1;
q2 := c1;
END_FUNCTION_BLOCK

(* POU EQUIP_TYPE_10, ST *)
FUNCTION_BLOCK EQUIP_TYPE_10
VAR_INPUT
	i1:BOOL;
	i2:BOOL;
	r1:BOOL;
	s1:BOOL;
	s2:BOOL;
	s3:BOOL;
	s4:BOOL;
	s5:BOOL;

END_VAR
VAR_OUTPUT
	q1:BOOL;
	q2:BOOL;
	e1:BOOL;
END_VAR
VAR
END_VAR
q1 := i1;
q2 := i2;
END_FUNCTION_BLOCK

(* POU EQUIPMENT_SBR_AIRBLOWER, ST *)
FUNCTION_BLOCK EQUIPMENT_SBR_AIRBLOWER
VAR_INPUT
	sa1 : BOOL;
	sa2 : BOOL;
	sa3 : BOOL;
	sa4 : BOOL;
	sa5 : BOOL;

	sb1 : BOOL;
	sb2 : BOOL;
	sb3 : BOOL;
	sb4 : BOOL;
	sb5 : BOOL;

	sc1 : BOOL;
	sc2 : BOOL;
	sc3 : BOOL;
	sc4 : BOOL;
	sc5 : BOOL;
	req : INT;

END_VAR
VAR_OUTPUT
	q1 : BOOL;
	q2 : BOOL;
	q3 : BOOL;
END_VAR
VAR
END_VAR
q1 := q2 := q3 := req > 0;
END_FUNCTION_BLOCK

(* POU sludge_holding, ST *)
FUNCTION_BLOCK sludge_holding
VAR_INPUT
	i1A : BOOL;
	i1B : BOOL;
	i2A : BOOL;
	i2B : BOOL;
	i3A : BOOL;
	i3B : BOOL;
	i4 : BOOL;
	i5 : BOOL;
	i6 : BOOL;
	i7 : BOOL;
	ic1 : BOOL;
	ic2 : BOOL;
	s1 : BOOL;
	s2 : BOOL;
	s3 : BOOL;
	s4 : BOOL;
	s5 : BOOL;
	r1 : BOOL;


END_VAR
VAR_OUTPUT
	q1A : BOOL;
	q2A : BOOL;
	q1B : BOOL;
	q2B : BOOL;
	q3 : BOOL;
	q4 : BOOL;
	q5 : BOOL;
	q6 : BOOL;
	q7 : BOOL;
	q8 : BOOL;
	q9 : BOOL;
	q10 : BOOL;
	q11 : BOOL;
	q12 : BOOL;
	q13 : BOOL;
	q14 : BOOL;
	c1 : BOOL;
	e1 : BOOL;

END_VAR
VAR
	TON1 : TON;
	TOF1 : TOF;
END_VAR
q1A := NOT i1A;
q2A := i2A;

q1B := NOT i1B;
q2B := i2B;

(*single switch convention*)
q3 := ic1 AND s4;
q4 := ic2 AND s5;

(* t /ops *)
c1 := (i2A OR i2B OR c1) AND NOT ((NOT i1A AND NOT i2A) OR s1 OR s2 OR s3 OR i7);

TON1(IN:=i4 , PT:=T#3s , Q=> , ET=> );
(*single switch*)
q5 := c1;
q6 := c1 AND TON1.Q;
q7 := c1;
q8 := c1;
q9 := c1;

q10 := i5;
q11 := (NOT i6) AND r1;
e1 := (e1 OR i6) AND NOT r1;
q12 := i6;

TOF1(IN:=i6 , PT:=T#30s , Q=> , ET=> );
q14 := q13 := c1 AND TOF1.Q;
END_FUNCTION_BLOCK

(* POU tertiary_treatment_plant, ST *)
FUNCTION_BLOCK tertiary_treatment_plant
VAR_INPUT
	i1 : BOOL;
	i2 : BOOL;
	i3 : BOOL;
	i4 : BOOL;
	i5 : BOOL;
	i6 : BOOL;
	i7 : BOOL;
	s1 : BOOL;
	s2 : BOOL;
	s3 : BOOL;
	s4 : BOOL;
END_VAR
VAR_OUTPUT
	q1: BOOL;
	q2 : BOOL;
	q3 : BOOL;
	q4 : BOOL;
	q5 : BOOL;
	q6 : BOOL;
	q7 : BOOL;
	q8 : BOOL;
	q9 : BOOL;
	q10 : BOOL;
	q11 : BOOL;
	q12 : BOOL;
END_VAR
VAR
END_VAR
q1 := i3 (*OR i4*);
q2 := i1 OR i2;
q3:= NOT(s3 OR s4);
q4 := (s3 OR s4);
q5 := NOT(s3 OR s4);
q6 := (s3 OR s4);
q7 := NOT ( s1 OR s2);
q8 := (s1 OR s2);
q9:= NOT(s1 OR s2);
q10 := i5 AND (s1 OR s2);
q11 := i7 OR NOT(s1 OR s2);
q12 := NOT i6 AND (s1 OR s2);
END_FUNCTION_BLOCK

(* POU REUSE_WATER, ST *)
FUNCTION_BLOCK REUSE_WATER
VAR_INPUT
	i3: BOOL;
	i1: BOOL;
	i4: BOOL;
	i2: BOOL;
	i5: BOOL;
	i6: BOOL;
	p1: REAL;


END_VAR
VAR_OUTPUT
	q1: BOOL;
	q2: BOOL;
	q3: BOOL;
	q4: BOOL;
	q5: BOOL;
	q6: BOOL;
	q7: BOOL;
	q8: BOOL;
	q9: BOOL;
END_VAR
VAR
	m1: BOOL;
	e1: BOOL;
	TON1: TON;
	m2: BOOL;
	TON2: TON;
END_VAR
q1 := (p1 > 8) OR (NOT m1) OR e1 OR i3;
q2 := (p1 <= 6) AND m1;

q3:=(p1 > 6.4) OR (NOT m1) OR e1 OR i3;
q4 := (p1 <= 5.2) AND m1;

q5:=(p1 > 5.9) OR (NOT m1) OR e1 OR i3;
q6 := (p1 <= 4.7) AND m1;

TON1(IN:=((p1 < 3.5) AND m1) , PT:=T#5s , Q=>e1 , ET=> );
TON2(IN:=i1 , PT:=T#5s , Q=> , ET=> );
m2 := TON2.Q    (*(i2 OR m2) AND i1*);
m1 := i4 AND m2;

q7 := i6;
q8 := i5;

q9 := TRUE;
END_FUNCTION_BLOCK

(* POU Aerate_selector, ST *)
FUNCTION_BLOCK Aerate_selector
VAR_INPUT
	i1: BOOL;
	i2: BOOL;
	i3: BOOL;
	i4: BOOL;
END_VAR
VAR_OUTPUT
	q1: BOOL;
	q2: BOOL;
	q3: BOOL;
	q4: BOOL;
	c1: BOOL;
END_VAR
VAR
	ireactor: INT;
END_VAR
q1 := q2 := q3 := q4 := FALSE;

CASE ireactor OF
0:
	IF NOT i1 THEN
		ireactor := 1;
	END_IF
	q1 := TRUE;
1:
	IF NOT i2 THEN
		ireactor := 2;
	END_IF
	q2 := TRUE;
2:
	IF NOT i3 THEN
		ireactor := 3;
	END_IF
	q3 := TRUE;
3:
	IF NOT i4 THEN
		ireactor := 0;
	END_IF
	q4 := TRUE;
END_CASE

c1 := i1 OR i2 OR i3 OR i4;
END_FUNCTION_BLOCK
